Universal Robots PolyScope program: switch_120.urp

Program switch_120 (createdIn=3.2.19293 lastSavedIn=3.2.19293 directory=/programs installation=default robotSerialNumber=2015351391)
Calibrated DH parameters: a=[0.000352, -0.161198, -0.373486, 0.00005, 0.000049, 0]; d=[0.089268, 352.477598, -320.08558, -32.281492, 0.094939, 0.082518]; alpha=[1.570728, 0.001116, -0.003686, 1.571189, -1.570572, 0]; deltaTheta=[-0.000012, 1.181849, -1.491165, 0.309495, -0.000007, 0.000025]
Robot Program (runOnlyOnce=false motionType=MoveJ speed=1.047198 acceleration=1.396263 recalculateMotions=false)
  select_no :=  (valueSource=Operator message=Enter a number between 1 to 3: valueType=Integer)
  Switch expression=select_no
    Case (caseValue=1)
      Popup Message (haltProgram=false message=product 1)
    Case (caseValue=2)
      Popup Message (haltProgram=false message=product 2)
    Case (caseValue=3)
      Popup Message (haltProgram=false message=product 3)
    Case (caseValue=2147483647)
      Popup Message (haltProgram=false message=wrong product number)
